// TIA Portal V17 export
// export: Created 2024-06-25T12:57:18.6779714Z, ExportSetting WithDefaults, DisplayName Totally Integrated Automation Portal, DisplayVersion V17 Update 6, DisplayName TIA Portal Openness, DisplayVersion V17 Update 6, DisplayName TIA Portal Version Control Interface, DisplayVersion V17, DisplayName STEP 7 Professional, DisplayVersion V17 Update 6, DisplayName STEP 7 Safety, DisplayVersion V17 Update 6, DisplayName WinCC Advanced, DisplayVersion V17 Update 6
FUNCTION "Logica" : Void   // FC4, LAD
{ S7_Optimized_Access := 'TRUE' }
VERSION : 0.1
// stored: AutoNumber true, IsIECCheckEnabled false, SetENOAutomatically false, UDAEnableTagReadback false
BEGIN

REGION Network 1: M_MODO_OFF
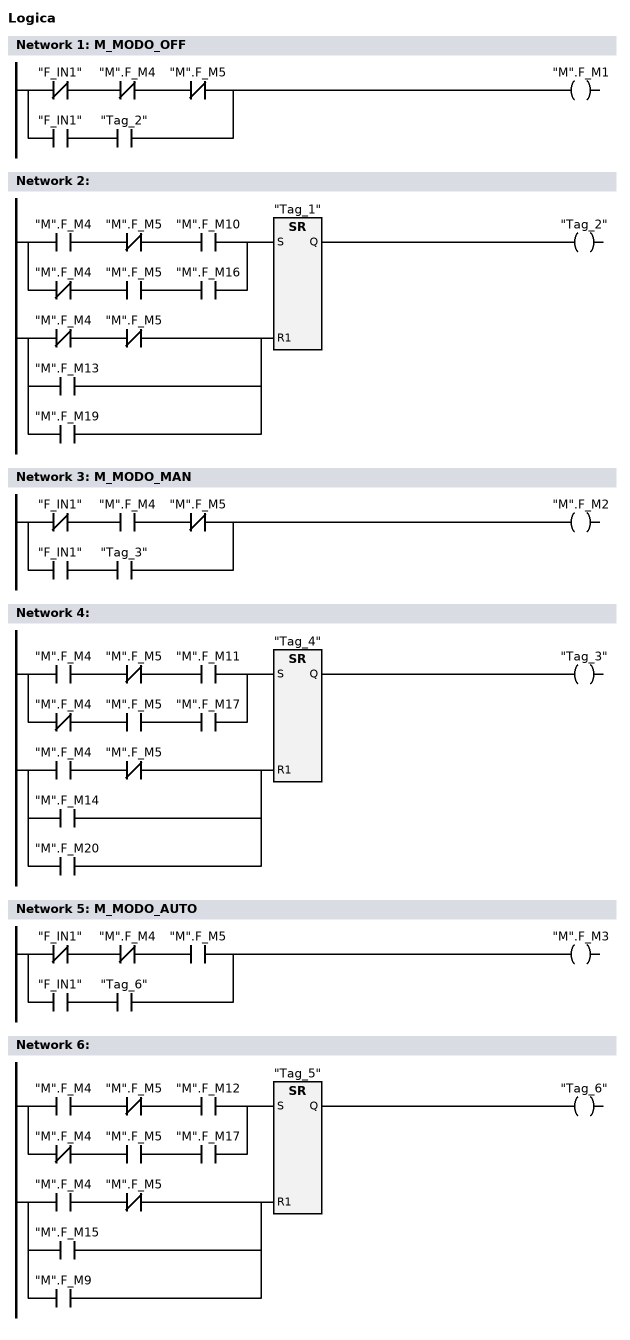
   RUNG wire#powerrail
      I_Contact( "F_IN1" )
      I_Contact( "M".F_M4 )
      I_Contact( "M".F_M5 )
      wire#w1
      Coil( "M".F_M1 )
   END_RUNG
   RUNG wire#powerrail
      Contact( "F_IN1" )
      Contact( "Tag_2" )
   END_RUNG wire#w1
   // the same network as SCL:
   "M".F_M1 := (NOT "F_IN1" AND NOT "M".F_M4 AND NOT "M".F_M5) OR ("F_IN1" AND "Tag_2");
END_REGION

REGION Network 2
   RUNG wire#powerrail
      Contact( "M".F_M4 )
      I_Contact( "M".F_M5 )
      Contact( "M".F_M10 )
      wire#w1
      S_SR(operand := "Tag_1", r1 := wire#w2)
      Coil( "Tag_2" )
   END_RUNG
   RUNG wire#powerrail
      I_Contact( "M".F_M4 )
      Contact( "M".F_M5 )
      Contact( "M".F_M16 )
   END_RUNG wire#w1
   RUNG wire#powerrail
      I_Contact( "M".F_M4 )
      I_Contact( "M".F_M5 )
   END_RUNG wire#w2
   RUNG wire#powerrail
      Contact( "M".F_M13 )
   END_RUNG wire#w2
   RUNG wire#powerrail
      Contact( "M".F_M19 )
   END_RUNG wire#w2
   // the same network as SCL:
   IF ("M".F_M4 AND NOT "M".F_M5 AND "M".F_M10) OR (NOT "M".F_M4 AND "M".F_M5 AND "M".F_M16) THEN
       "Tag_1" := TRUE;   // SR flip-flop
   END_IF;
   IF (NOT "M".F_M4 AND NOT "M".F_M5) OR "M".F_M13 OR "M".F_M19 THEN "Tag_1" := FALSE; END_IF;
   "Tag_2" := "Tag_1";
END_REGION

REGION Network 3: M_MODO_MAN
   RUNG wire#powerrail
      I_Contact( "F_IN1" )
      Contact( "M".F_M4 )
      I_Contact( "M".F_M5 )
      wire#w1
      Coil( "M".F_M2 )
   END_RUNG
   RUNG wire#powerrail
      Contact( "F_IN1" )
      Contact( "Tag_3" )
   END_RUNG wire#w1
   // the same network as SCL:
   "M".F_M2 := (NOT "F_IN1" AND "M".F_M4 AND NOT "M".F_M5) OR ("F_IN1" AND "Tag_3");
END_REGION

REGION Network 4
   RUNG wire#powerrail
      Contact( "M".F_M4 )
      I_Contact( "M".F_M5 )
      Contact( "M".F_M11 )
      wire#w1
      S_SR(operand := "Tag_4", r1 := wire#w2)
      Coil( "Tag_3" )
   END_RUNG
   RUNG wire#powerrail
      I_Contact( "M".F_M4 )
      Contact( "M".F_M5 )
      Contact( "M".F_M17 )
   END_RUNG wire#w1
   RUNG wire#powerrail
      Contact( "M".F_M4 )
      I_Contact( "M".F_M5 )
   END_RUNG wire#w2
   RUNG wire#powerrail
      Contact( "M".F_M14 )
   END_RUNG wire#w2
   RUNG wire#powerrail
      Contact( "M".F_M20 )
   END_RUNG wire#w2
   // the same network as SCL:
   IF ("M".F_M4 AND NOT "M".F_M5 AND "M".F_M11) OR (NOT "M".F_M4 AND "M".F_M5 AND "M".F_M17) THEN
       "Tag_4" := TRUE;   // SR flip-flop
   END_IF;
   IF ("M".F_M4 AND NOT "M".F_M5) OR "M".F_M14 OR "M".F_M20 THEN "Tag_4" := FALSE; END_IF;
   "Tag_3" := "Tag_4";
END_REGION

REGION Network 5: M_MODO_AUTO
   RUNG wire#powerrail
      I_Contact( "F_IN1" )
      I_Contact( "M".F_M4 )
      Contact( "M".F_M5 )
      wire#w1
      Coil( "M".F_M3 )
   END_RUNG
   RUNG wire#powerrail
      Contact( "F_IN1" )
      Contact( "Tag_6" )
   END_RUNG wire#w1
   // the same network as SCL:
   "M".F_M3 := (NOT "F_IN1" AND NOT "M".F_M4 AND "M".F_M5) OR ("F_IN1" AND "Tag_6");
END_REGION

REGION Network 6
   RUNG wire#powerrail
      Contact( "M".F_M4 )
      I_Contact( "M".F_M5 )
      Contact( "M".F_M12 )
      wire#w1
      S_SR(operand := "Tag_5", r1 := wire#w2)
      Coil( "Tag_6" )
   END_RUNG
   RUNG wire#powerrail
      I_Contact( "M".F_M4 )
      Contact( "M".F_M5 )
      Contact( "M".F_M17 )
   END_RUNG wire#w1
   RUNG wire#powerrail
      Contact( "M".F_M4 )
      I_Contact( "M".F_M5 )
   END_RUNG wire#w2
   RUNG wire#powerrail
      Contact( "M".F_M15 )
   END_RUNG wire#w2
   RUNG wire#powerrail
      Contact( "M".F_M9 )
   END_RUNG wire#w2
   // the same network as SCL:
   IF ("M".F_M4 AND NOT "M".F_M5 AND "M".F_M12) OR (NOT "M".F_M4 AND "M".F_M5 AND "M".F_M17) THEN
       "Tag_5" := TRUE;   // SR flip-flop
   END_IF;
   IF ("M".F_M4 AND NOT "M".F_M5) OR "M".F_M15 OR "M".F_M9 THEN "Tag_5" := FALSE; END_IF;
   "Tag_6" := "Tag_5";
END_REGION
END_FUNCTION
